Staubli VAL3: isInList.pgx

program isInList(string x_sInputString (dimensions=1), string& x_sItemList[] (dimensions=1), bool& x_bIsInList[] (dimensions=1))
  local num l_i
begin
  // This program checks if the input string  belongs to the
  // Stringlist item
  //
  //
  // Created 12-10-07                                   C.CURRIVAND
  //----------------------------------------------------------------
  l_i=0
  x_bIsInList=false
  while (l_i<size(x_sItemList) and !x_bIsInList)
    x_bIsInList=(x_sInputString==x_sItemList[l_i])
    l_i=l_i+1
  endWhile
end
